RESOURCE_TYPE TrainGate
  (* Standard: 61499-2 *)
  (* Version 0.1, 2017-00-23, hpea485, UOA *)
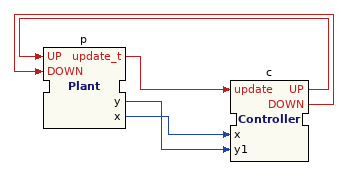
  FBS
    p : Plant;
    c : Controller;
  END_FBS
  EVENT_CONNECTIONS
    p.update_t TO c.update;
    c.UP TO p.UP;
    c.DOWN TO p.DOWN;
  END_CONNECTIONS
  DATA_CONNECTIONS
    p.y TO c.y1;
    p.x TO c.x;
  END_CONNECTIONS
END_RESOURCE_TYPE
